FUNCTION_BLOCK FB_HomeableEncAxis EXTENDS FB_HomeableAxis
VAR_INPUT
END_VAR
VAR_OUTPUT
END_VAR
VAR
	fbEncWait : TON;
	bEnableLatchC AT %Q*: BOOL;
END_VAR

	IF bFirstCycle THEN
		piHomeSensor.Description := 'Encoder C track';
	END_IF

	SUPER^();

METHOD PROTECTED StateHoming : BOOL // Unit is performing action 1
VAR_INPUT
END_VAR
IF NOT fbMcHome.Error THEN // no error behavior

//Home
	fbMcHome(		Execute 	:= TRUE,
					Axis		:= AxisRef,
					HomingMode	:= MC_DefaultHoming,
					bCalibratioNCam		:= piHomeSensor.Value);
	
	bEnableLatchC := TRUE;
	fbEncWait(IN := piHomeSensor.Value, PT:= T#1000MS);
	bEnableLatchC R= fbEncWait.Q;
	
	IF fbMcHome.Done THEN
		iStepGeneral := 50;
		fbMcHome(	Execute 	:= FALSE,
					Axis		:= AxisRef,
					HomingMode	:= MC_DefaultHoming,
					bCalibratioNCam		:= piHomeSensor.Value);
		bEnableLatchC := FALSE;
	END_IF

ELSE // error behavior
	fbMcHome(		Execute 	:= FALSE,
					Axis		:= AxisRef,
					HomingMode	:= MC_DefaultHoming,
					bCalibratioNCam		:= piHomeSensor.Value);
	
	bEnableLatchC := FALSE;
	bError		:= TRUE;
	iErrorID 	:= fbMcHome.ErrorID;
END_IF
END_METHOD

END_FUNCTION_BLOCK

(* stored: Version 1.1.0.1, ProductVersion 3.1.4024.9
   POU FB_HomeableEncAxis: Id {47e1576d-a738-47ef-bdf3-20a64e9797eb}, SpecialFunc None
   Method StateHoming: Id {30964498-4c80-41dd-942a-8170f783a822} *)
